{attribute 'GeneratedUsingTerminal: EP2328-1061-0016'}
{attribute addProperty BoxType "EP2328-1061-0016"}
{attribute addProperty Id "InputAT %I*BOOL1"}
{attribute addProperty CRC "2198356929"}
{attribute addProperty Size "1"}
TYPE DI_X02_Pin2_Input_830843C1 :
STRUCT
	{attribute addProperty Name "Input"}
	Input AT %I* : BOOL;
END_STRUCT
END_TYPE

(* stored: Version 1.2.0.0, ProductVersion 3.1.4024.9
   DUT DI_X02_Pin2_Input_830843C1: Id {e7fe2204-2716-490b-8a4a-d4280e4a7411} *)
